Universal Robots PolyScope program: stacking_p1.urp

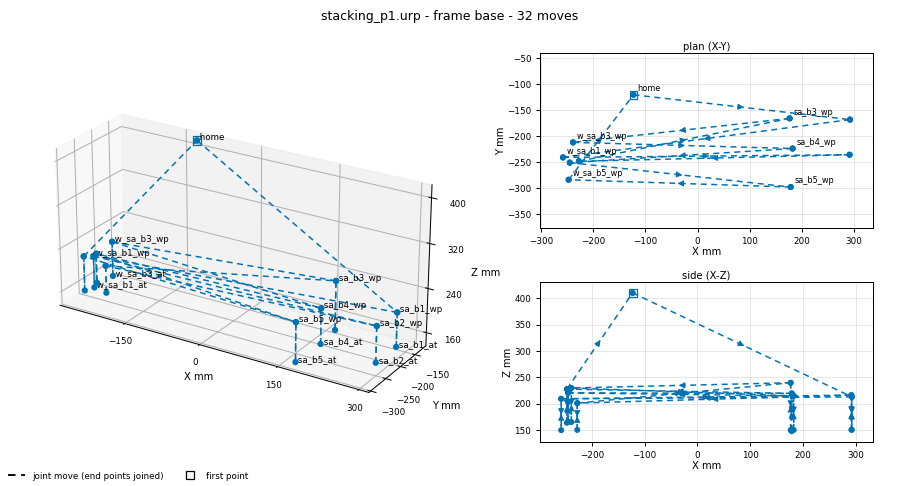
[picture p0: tool path of stacking_p1.urp in frame base, 32 of 32 moves have a stored position in this frame; points joined in program order, loops and branches not executed]
Program stacking_p1 (installation=default directory=/programs/ITER createdIn=5.3.1.64192 lastSavedIn=5.3.1.64192 robotSerialNumber=20195300365)
Calibrated DH parameters: a=[-0.000093, -0.190649, -0.212673, 0.000091, -0.000205, 0]; d=[0.151591, 44.061648, -42.488068, -1.442789, 0.085322, 0.091911]; alpha=[1.570082, -0.003447, 0.007513, 1.572293, -1.571904, 0]; deltaTheta=[0, -0.672656, 0.728185, -0.055522, 0.000005, 0]
Robot Program (runOnlyOnce=true)
  URCap Gripper Activate (Robotiq_Grippers, Robotiq Inc.) dataModel(ResetAndActivateKey=false)
  URCap Gripper (Robotiq_Grippers, Robotiq Inc.) dataModel(position=50.19607843137255, force=100.0, speed=100.0, positionInDouble=50.19607843137255, forceInDouble=100.0, speedInDouble=100.0, slaveIds=[9], blocking=true)
  MoveJ speed 60 deg/s, acceleration 80 deg/s^2 (useActiveTCP=true) feature=Base
    Waypoint home: TCP in base x=-122.938 y=-120.383 z=410.034 mm, rx=2.2731 ry=2.1658 rz=-0.0264 rad; joints [-85.881, -57.164, -80.451, -131.628, 89.647, -263.137] deg
  Folder Stack A
    MoveJ speed 60 deg/s, acceleration 80 deg/s^2 (useActiveTCP=true) feature=Base
      Waypoint sa_b1_wp: TCP in base x=292.404 y=-167.975 z=213.105 mm, rx=2.2724 ry=2.1125 rz=-0.0265 rad; joints [-6.643, -96.999, -108.294, -63.598, 88.105, -182.097] deg
      Waypoint sa_b1_at: TCP in base x=292.4 y=-167.967 z=150.758 mm, rx=2.2724 ry=2.1125 rz=-0.0265 rad; joints [-6.665, -105.883, -117.26, -45.753, 88.016, -182.03] deg
      URCap Gripper (Robotiq_Grippers, Robotiq Inc.) dataModel(position=100.0, force=100.0, speed=100.0, positionInDouble=100.0, forceInDouble=100.0, speedInDouble=100.0, slaveIds=[9], blocking=true)
      Waypoint sa_b1_wp: TCP in base x=292.404 y=-167.975 z=213.105 mm, rx=2.2724 ry=2.1125 rz=-0.0265 rad; joints [-6.643, -96.999, -108.294, -63.598, 88.105, -182.097] deg
      Waypoint w_sa_b1_wp: TCP in base x=-258.271 y=-240.499 z=209.476 mm, rx=3.1151 ry=-0.0825 rz=0.0204 rad; joints [-115.862, -101.636, -103.759, -63.52, 91.564, -202.433] deg
      Waypoint w_sa_b1_at: TCP in base x=-258.276 y=-240.491 z=150.031 mm, rx=3.1151 ry=-0.0827 rz=0.0205 rad; joints [-115.884, -109.689, -111.896, -47.33, 91.487, -202.37] deg
      URCap Gripper (Robotiq_Grippers, Robotiq Inc.) dataModel(position=50.19607843137255, force=100.0, speed=100.0, positionInDouble=50.19607843137255, forceInDouble=100.0, speedInDouble=100.0, slaveIds=[9], blocking=true)
      Waypoint w_sa_b1_wp: TCP in base x=-258.271 y=-240.499 z=209.476 mm, rx=3.1151 ry=-0.0825 rz=0.0204 rad; joints [-115.862, -101.636, -103.759, -63.52, 91.564, -202.433] deg
    MoveJ speed 60 deg/s, acceleration 80 deg/s^2 (useActiveTCP=true) feature=Base
      Waypoint sa_b2_wp: TCP in base x=291.521 y=-235.36 z=216.434 mm, rx=-2.2136 ry=-2.2083 rz=0.0077 rad; joints [-18.698, -106.327, -94.779, -69.718, 90.416, -198.233] deg
      Waypoint sa_b2_at: TCP in base x=291.522 y=-235.352 z=150.683 mm, rx=-2.2136 ry=-2.2083 rz=0.0078 rad; joints [-18.72, -114.004, -103.962, -52.861, 90.345, -198.164] deg
      URCap Gripper (Robotiq_Grippers, Robotiq Inc.) dataModel(position=100.0, force=100.0, speed=100.0, positionInDouble=100.0, forceInDouble=100.0, speedInDouble=100.0, slaveIds=[9], blocking=true)
      Waypoint sa_b2_wp: TCP in base x=291.521 y=-235.36 z=216.434 mm, rx=-2.2136 ry=-2.2083 rz=0.0077 rad; joints [-18.698, -106.327, -94.779, -69.718, 90.416, -198.233] deg
      Waypoint w_sa_b2_wp: TCP in base x=-227.79 y=-247.903 z=201.3 mm, rx=-3.1116 ry=0.1046 rz=-0.0512 rad; joints [-110.33, -99.289, -107.723, -65.024, 91.583, -196.119] deg
      Waypoint w_sa_b2_at: TCP in base x=-227.812 y=-247.879 z=150.535 mm, rx=-3.1115 ry=0.1048 rz=-0.0512 rad; joints [-110.354, -106.436, -114.862, -50.742, 91.515, -196.061] deg
      URCap Gripper (Robotiq_Grippers, Robotiq Inc.) dataModel(position=50.19607843137255, force=100.0, speed=100.0, positionInDouble=50.19607843137255, forceInDouble=100.0, speedInDouble=100.0, slaveIds=[9], blocking=true)
      Waypoint w_sa_b2_wp: TCP in base x=-227.79 y=-247.903 z=201.3 mm, rx=-3.1116 ry=0.1046 rz=-0.0512 rad; joints [-110.33, -99.289, -107.723, -65.024, 91.583, -196.119] deg
    MoveJ speed 60 deg/s, acceleration 80 deg/s^2 (useActiveTCP=true) feature=Base
      Waypoint sa_b3_wp: TCP in base x=176.502 y=-165.594 z=239.893 mm, rx=2.2432 ry=2.1833 rz=0.0345 rad; joints [-11.13, -68.37, -125.032, -75.288, 91.077, 170.788] deg
      Waypoint sa_b3_at: TCP in base x=176.504 y=-165.593 z=150.238 mm, rx=2.2432 ry=2.1834 rz=0.0344 rad; joints [-11.187, -82.894, -143.393, -42.404, 90.919, 170.923] deg
      URCap Gripper (Robotiq_Grippers, Robotiq Inc.) dataModel(position=100.0, force=100.0, speed=100.0, positionInDouble=100.0, forceInDouble=100.0, speedInDouble=100.0, slaveIds=[9], blocking=true)
      Waypoint sa_b3_wp: TCP in base x=176.502 y=-165.594 z=239.893 mm, rx=2.2432 ry=2.1833 rz=0.0345 rad; joints [-11.13, -68.37, -125.032, -75.288, 91.077, 170.788] deg
      Waypoint w_sa_b3_wp: TCP in base x=-238.992 y=-211.647 z=229.952 mm, rx=-2.2294 ry=-2.1837 rz=0.0163 rad; joints [-114.115, -91.23, -109.253, -69.342, 88.995, -292.563] deg
      Waypoint w_sa_b3_at: TCP in base x=-238.971 y=-211.668 z=165.415 mm, rx=-2.2293 ry=-2.1838 rz=0.0164 rad; joints [-114.137, -99.517, -120.016, -50.29, 88.907, -292.484] deg
      URCap Gripper (Robotiq_Grippers, Robotiq Inc.) dataModel(position=50.19607843137255, force=100.0, speed=100.0, positionInDouble=50.19607843137255, forceInDouble=100.0, speedInDouble=100.0, slaveIds=[9], blocking=true)
      Waypoint w_sa_b3_wp: TCP in base x=-238.992 y=-211.647 z=229.952 mm, rx=-2.2294 ry=-2.1837 rz=0.0163 rad; joints [-114.115, -91.23, -109.253, -69.342, 88.995, -292.563] deg
    MoveJ speed 60 deg/s, acceleration 80 deg/s^2 (useActiveTCP=true) feature=Base
      Waypoint sa_b4_wp: TCP in base x=182.289 y=-223.443 z=214.982 mm, rx=2.2444 ry=2.1711 rz=-0.0785 rad; joints [-23.025, -84.233, -120.167, -65.731, 87.284, -200.715] deg
      Waypoint sa_b4_at: TCP in base x=182.287 y=-223.437 z=150.399 mm, rx=2.2444 ry=2.1711 rz=-0.0784 rad; joints [-23.054, -94.883, -130.899, -44.355, 87.172, -200.631] deg
      URCap Gripper (Robotiq_Grippers, Robotiq Inc.) dataModel(position=100.0, force=100.0, speed=100.0, positionInDouble=100.0, forceInDouble=100.0, speedInDouble=100.0, slaveIds=[9], blocking=true)
      Waypoint sa_b4_wp: TCP in base x=182.289 y=-223.443 z=214.982 mm, rx=2.2444 ry=2.1711 rz=-0.0785 rad; joints [-23.025, -84.233, -120.167, -65.731, 87.284, -200.715] deg
      Waypoint w_sa_b4_wp: TCP in base x=-245.189 y=-250.465 z=220.693 mm, rx=2.2499 ry=2.1886 rz=-0.0042 rad; joints [-112.717, -99.979, -102.147, -67.604, 90.389, -290.778] deg
      Waypoint w_sa_b4_at: TCP in base x=-245.197 y=-250.444 z=165.926 mm, rx=2.25 ry=2.1885 rz=-0.0041 rad; joints [-112.742, -106.561, -110.516, -52.658, 90.325, -290.716] deg
      URCap Gripper (Robotiq_Grippers, Robotiq Inc.) dataModel(position=50.19607843137255, force=100.0, speed=100.0, positionInDouble=50.19607843137255, forceInDouble=100.0, speedInDouble=100.0, slaveIds=[9], blocking=true)
      Waypoint w_sa_b4_wp: TCP in base x=-245.189 y=-250.465 z=220.693 mm, rx=2.2499 ry=2.1886 rz=-0.0042 rad; joints [-112.717, -99.979, -102.147, -67.604, 90.389, -290.778] deg
    MoveJ speed 60 deg/s, acceleration 80 deg/s^2 (useActiveTCP=true) feature=Base
      Waypoint sa_b5_wp: TCP in base x=178.546 y=-297.407 z=219.75 mm, rx=-2.2213 ry=-2.2161 rz=0.0093 rad; joints [-37, -99.244, -103.103, -67.859, 89.998, -216.508] deg
      Waypoint sa_b5_at: TCP in base x=178.517 y=-297.407 z=148.098 mm, rx=-2.2213 ry=-2.2161 rz=0.0094 rad; joints [-37.029, -108.645, -113.454, -48.11, 89.904, -216.432] deg
      URCap Gripper (Robotiq_Grippers, Robotiq Inc.) dataModel(position=100.0, force=100.0, speed=100.0, positionInDouble=100.0, forceInDouble=100.0, speedInDouble=100.0, slaveIds=[9], blocking=true)
      Waypoint sa_b5_wp: TCP in base x=178.546 y=-297.407 z=219.75 mm, rx=-2.2213 ry=-2.2161 rz=0.0093 rad; joints [-37, -99.244, -103.103, -67.859, 89.998, -216.508] deg
      Waypoint w_sa_b5_wp: TCP in base x=-247.393 y=-283.334 z=227.844 mm, rx=2.2495 ry=2.1402 rz=-0.0127 rad; joints [-111.4, -105.454, -93.637, -69.526, 91.99, -288.199] deg
      Waypoint w_sa_b5_at: TCP in base x=-247.399 y=-283.319 z=164.004 mm, rx=2.2496 ry=2.1402 rz=-0.0126 rad; joints [-111.426, -112.371, -103.175, -53.072, 91.924, -288.131] deg
      URCap Gripper (Robotiq_Grippers, Robotiq Inc.) dataModel(position=50.19607843137255, force=100.0, speed=100.0, positionInDouble=50.19607843137255, forceInDouble=100.0, speedInDouble=100.0, slaveIds=[9], blocking=true)
      Waypoint w_sa_b5_wp: TCP in base x=-247.393 y=-283.334 z=227.844 mm, rx=2.2495 ry=2.1402 rz=-0.0127 rad; joints [-111.4, -105.454, -93.637, -69.526, 91.99, -288.199] deg
  MoveJ speed 60 deg/s, acceleration 80 deg/s^2 (useActiveTCP=true) feature=Base
    Waypoint home: TCP in base x=-122.938 y=-120.383 z=410.034 mm, rx=2.2731 ry=2.1658 rz=-0.0264 rad; joints [-85.881, -57.164, -80.451, -131.628, 89.647, -263.137] deg
